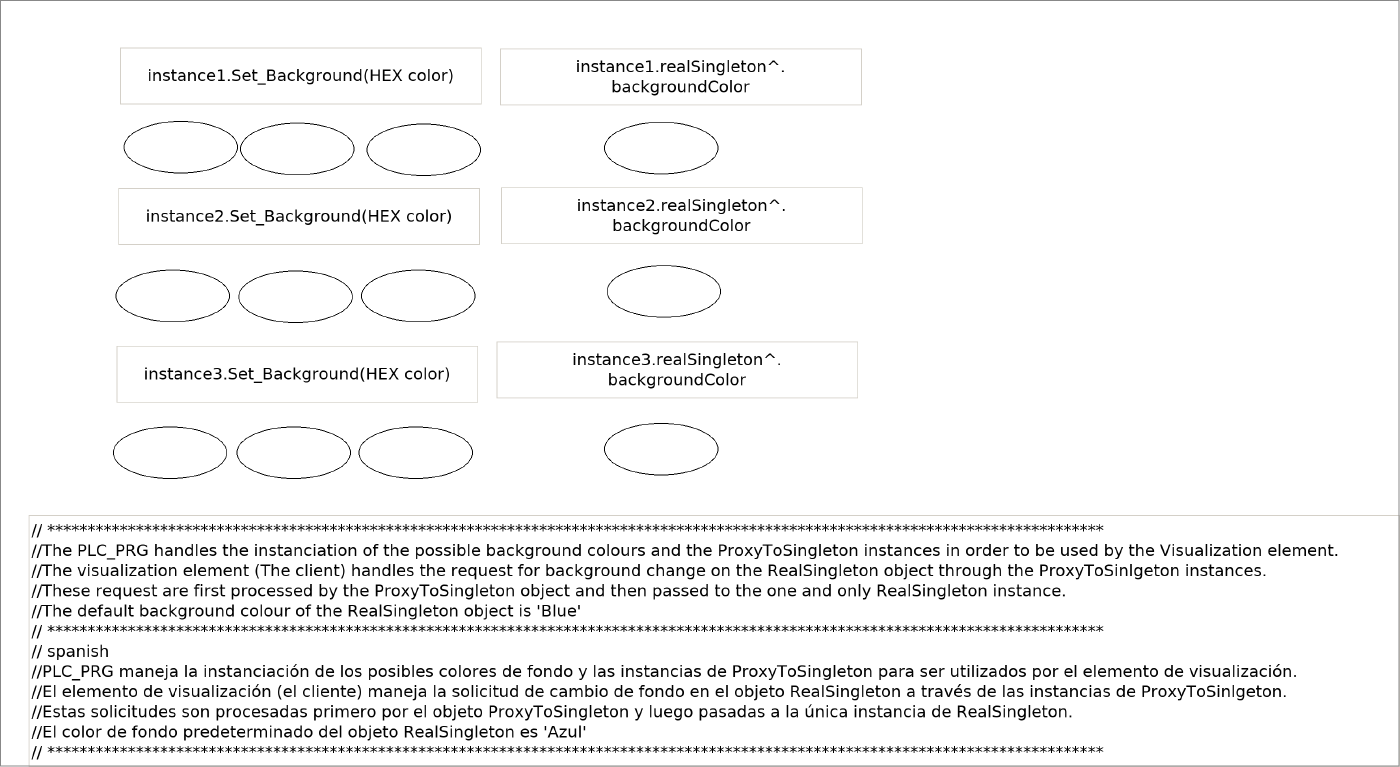
VISUALIZATION Visualization  // 1562x856
    Textfield (134,53 403x63), "instance1.Set_Background(HEX color)"
    Textfield (558,54 403x63), "instance1.realSingleton^. backgroundColor"
    Textfield (132,210 403x63), "instance2.Set_Background(HEX color)"
    Textfield (130,386 403x63), "instance3.Set_Background(HEX color)"
    Textfield (559,209 403x63), "instance2.realSingleton^. backgroundColor"
    Textfield (554,381 403x63), "instance3.realSingleton^. backgroundColor"
    Ellipse (138,135 127x58), colour variable: PLC_PRG.dwBlue
        OnMouseClick: execute {
            //PLC_PRG.instance1.Set_Background(newBackground:=PLC_PRG.dwBlue);
            PLC_PRG.eInstance1 := E_Color.Blue;
        }
    Ellipse (409,138 127x58), colour variable: PLC_PRG.dwYellow
        OnMouseClick: execute {
            //PLC_PRG.instance1.Set_Background(newBackground:=PLC_PRG.dwYellow);
            PLC_PRG.eInstance1 := E_Color.Yellow;
        }
    Ellipse (268,137 127x58), colour variable: PLC_PRG.dwGreen
        OnMouseClick: execute {
            //PLC_PRG.instance1.Set_Background(newBackground:=PLC_PRG.dwGreen);
            PLC_PRG.eInstance1 := E_Color.Green;
        }
    Ellipse (129,301 127x58), colour variable: PLC_PRG.dwBlue
        OnMouseClick: execute {
            //PLC_PRG.instance2.Set_Background(PLC_PRG.dwBlue);
            PLC_PRG.eInstance2 := E_Color.Blue;
        }
    Ellipse (403,301 127x58), colour variable: PLC_PRG.dwYellow
        OnMouseClick: execute {
            //PLC_PRG.instance2.Set_Background(PLC_PRG.dwYellow);
            PLC_PRG.eInstance2 := E_Color.Yellow;
        }
    Ellipse (266,302 127x58), colour variable: PLC_PRG.dwGreen
        OnMouseClick: execute {
            //PLC_PRG.instance2.Set_Background(PLC_PRG.dwGreen);
            PLC_PRG.eInstance2 := E_Color.Green;
        }
    Ellipse (126,476 127x58), colour variable: PLC_PRG.dwBlue
        OnMouseClick: execute {
            //PLC_PRG.instance3.Set_Background(PLC_PRG.dwBlue);
            PLC_PRG.eInstance3 := E_Color.Blue;
        }
    Ellipse (400,476 127x58), colour variable: PLC_PRG.dwYellow
        OnMouseClick: execute {
            //PLC_PRG.instance3.Set_Background(PLC_PRG.dwYellow);
            PLC_PRG.eInstance3 := E_Color.Yellow;
        }
    Ellipse (264,476 127x58), colour variable: PLC_PRG.dwGreen
        OnMouseClick: execute {
            //PLC_PRG.instance3.Set_Background(PLC_PRG.dwGreen);
            PLC_PRG.eInstance3 := E_Color.Green;
        }
    Ellipse (674,472 127x58), colour variable: PLC_PRG.instance3.realSingleton^.backgroundColour
    Ellipse (677,296 127x58), colour variable: PLC_PRG.instance2.realSingleton^.backgroundColour
    Ellipse (674,136 127x58), colour variable: PLC_PRG.instance1.realSingleton^.backgroundColour
    Textfield (32,575 1530x281), "// *********************************************************************************************************************************** //The PLC_PRG handles the instanciation of the possible background colours and the ProxyToSingleton instances in order to be used by the Visualization element. //The visualization element (The client) handles the request for background change on the RealSingleton object through the ProxyToSinlgeton instances. //These request are first processed by the ProxyToSingleton object and then passed to the one and only RealSingleton instance. //The default background colour of the RealSingleton object is 'Blue' // *********************************************************************************************************************************** // spanish //PLC_PRG maneja la instanciación de los posibles colores de fondo y las instancias de ProxyToSingleton para ser utilizados por el elemento de visualización. //El elemento de visualización (el cliente) maneja la solicitud de cambio de fondo en el objeto RealSingleton a través de las instancias de ProxyToSinlgeton. //Estas solicitudes son procesadas primero por el objeto ProxyToSingleton y luego pasadas a la única instancia de RealSingleton. //El color de fondo predeterminado del objeto RealSingleton es 'Azul' // ***********************************************************************************************************************************"
END_VISUALIZATION

(* stored: Version 1.1.0.1, ProductVersion 3.1.4024.12
   Visu Visualization: Id {794e636f-d6f7-4023-a5ff-448d003ef8e3} *)
